// Type alias for represeting size or capacity.
TYPE T_Size : UDINT; END_TYPE

(* stored: Version 1.1.0.1
   DUT T_Size: Id {4ee04fa1-0d24-065d-2124-018c78d976e8} *)
